TEXTLIST TextList_TwinSAFE_Group_State
  1 = 'RUN'
  2 = 'STOP'
  4 = 'ERROR'
  5 = 'RESET'
  6 = 'START'
  7 = 'STOPERROR'
  16 = 'DEACTIVE'
  17 = 'WAITCOMERROR'
   = ''
END_TEXTLIST

(* stored: Version 1.1.0.1, ProductVersion 3.1.4024.11
   TextList TextList_TwinSAFE_Group_State: Id {d1db6a7a-549c-4952-9a68-2d76bd2bba0f} *)
